PROGRAM MAIN
VAR
	bRunning : BOOL;
END_VAR

IF GVL.bStart THEN
	GVL.nCount := GVL.nCount + 1;
	//GVL.bStart := FALSE;
	bRunning := TRUE;
ELSE
	bRunning := FALSE;
END_IF

END_PROGRAM

(* stored: Version 1.1.0.1, ProductVersion 3.1.4024.16
   POU MAIN: Id {8a99b40e-55e8-44e4-bd59-a31b61aa9f2d}, SpecialFunc None *)
